{attribute 'linkalways'} 
{attribute 'no_explicit_call' := 'This FB is a CLASS and must be accessed using methods or properties'}
{attribute 'enable_dynamic_creation'}
FUNCTION_BLOCK FINAL OR_UDINT EXTENDS Node
VAR
	in1 : _UDINT(0);
	in2 : _UDINT(0);
	out : _UDINT(0);
END_VAR

METHOD PUBLIC Clone : I_Node
VAR
	pNode : POINTER TO OR_UDINT;
END_VAR
pNode := __NEW(OR_UDINT);
Clone := pNode^;
END_METHOD

METHOD FB_init : BOOL
VAR_INPUT
	bInitRetains : BOOL; // if TRUE, the retain variables are initialized (warm start / cold start)
	bInCopyCode : BOOL;  // if TRUE, the instance afterwards gets moved into the copy code (online change)
END_VAR
AddInput('in1',THIS^.in1);
AddInput('in2',THIS^.in2);
AddOutput('out', THIS^.out);
END_METHOD

METHOD PROTECTED OnExecute
VAR
END_VAR
out.Value := in1.Value OR in2.Value;
END_METHOD

END_FUNCTION_BLOCK

(* stored: Version 1.1.0.1, ProductVersion 3.1.4024.15
   POU OR_UDINT: Id {d07927f5-8080-4bd6-8ef4-8115782dfdc5}, SpecialFunc None
   Folder Constructor: Id {593489c4-c094-4c8e-ab9a-5f2923b3080d}
   Method Clone: Id {bae71af4-b2c0-4fc8-abc8-d99295ab7e9a}
   Method FB_init: Id {78c1839e-305c-43a9-b2fe-1d4abf229ae6}
   Method OnExecute: Id {71f85a83-da33-4b38-87d8-03ab0d8f9c1d} *)
